# EPICS autosave request: iocBoot/ioc13idc_linux/Galil_auto_positions.req
file "CARS_24_motor_positions.req", P=$(P)
file "CARS_motor_positions.req",         P=$(P), M=m57
file "CARS_motor_positions.req",         P=$(P), M=m58
file "CARS_motor_positions.req",         P=$(P), M=m59
file "CARS_motor_positions.req",         P=$(P), M=m60
file "CARS_motor_positions.req",         P=$(P), M=m61
file "CARS_motor_positions.req",         P=$(P), M=m62
file "CARS_motor_positions.req",         P=$(P), M=m63
file "CARS_motor_positions.req",         P=$(P), M=m64
